(* Logix 5000 project; controller RN21_Architecture 1769-L16ER-BB1B rev 35.11; software revision 35.00; part 4 of 9 *)
(* tags used below, declared in another part *)
   AUDSrc : UDT_Audit;
   RN21_AUD_BAT_NTrig : DINT[4];
   RN21_AUD_BAT_PTrig : DINT[4];
   RN21_AUD_NEG_ONS : BOOL[128];
   RN21_AUD_POS_ONS : BOOL[128];
   RN21_Map_BAT : BOOL[32];
   RN21_MapBAT_OB : BOOL[128];
(* MainProgram, continued *)

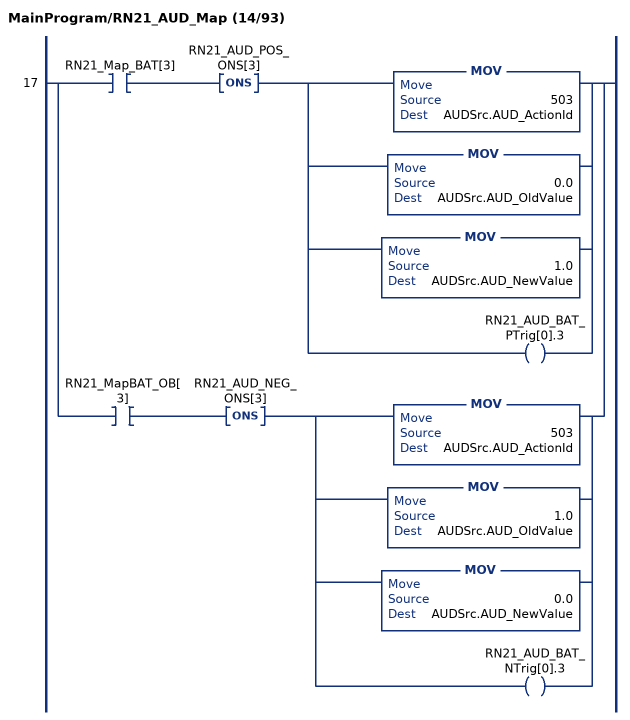
   [picture p96: MainProgram/RN21_AUD_Map rungs 17-17]
   17: [XIC(RN21_Map_BAT[3]) ONS(RN21_AUD_POS_ONS[3]) [MOV(503,AUDSrc.AUD_ActionId) ,MOV(0.0,AUDSrc.AUD_OldValue) ,MOV(1.0,AUDSrc.AUD_NewValue) ,OTE(RN21_AUD_BAT_PTrig[0].3) ] ,XIC(RN21_MapBAT_OB[3]) ONS(RN21_AUD_NEG_ONS[3]) [MOV(503,AUDSrc.AUD_ActionId) ,MOV(1.0,AUDSrc.AUD_OldValue) ,MOV(0.0,AUDSrc.AUD_NewValue) ,OTE(RN21_AUD_BAT_NTrig[0].3) ] ];
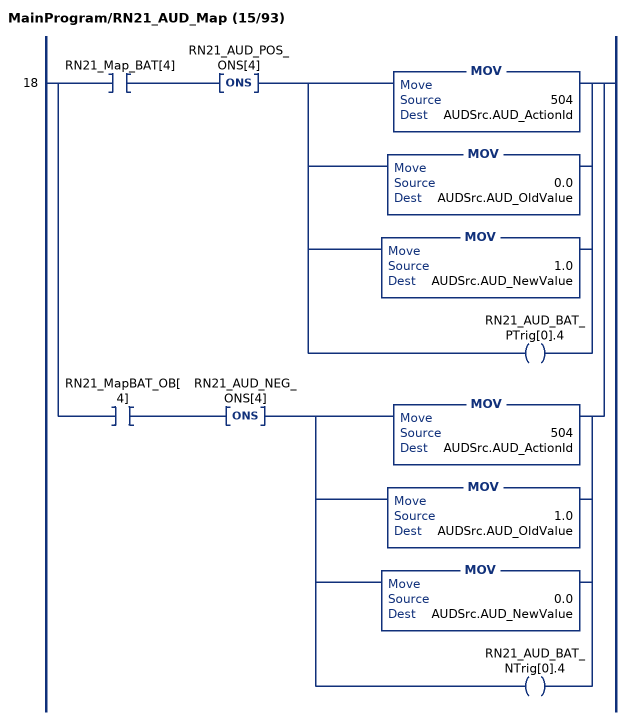
   18: [XIC(RN21_Map_BAT[4]) ONS(RN21_AUD_POS_ONS[4]) [MOV(504,AUDSrc.AUD_ActionId) ,MOV(0.0,AUDSrc.AUD_OldValue) ,MOV(1.0,AUDSrc.AUD_NewValue) ,OTE(RN21_AUD_BAT_PTrig[0].4) ] ,XIC(RN21_MapBAT_OB[4]) ONS(RN21_AUD_NEG_ONS[4]) [MOV(504,AUDSrc.AUD_ActionId) ,MOV(1.0,AUDSrc.AUD_OldValue) ,MOV(0.0,AUDSrc.AUD_NewValue) ,OTE(RN21_AUD_BAT_NTrig[0].4) ] ];
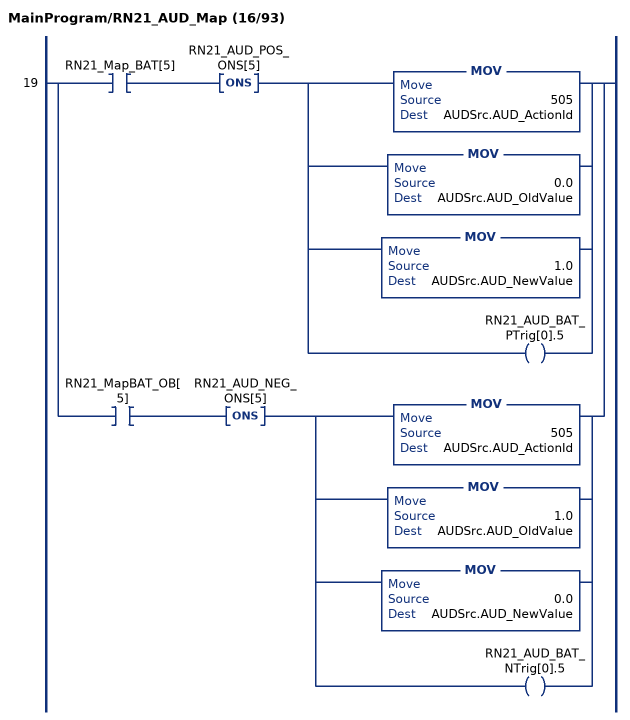
   19: [XIC(RN21_Map_BAT[5]) ONS(RN21_AUD_POS_ONS[5]) [MOV(505,AUDSrc.AUD_ActionId) ,MOV(0.0,AUDSrc.AUD_OldValue) ,MOV(1.0,AUDSrc.AUD_NewValue) ,OTE(RN21_AUD_BAT_PTrig[0].5) ] ,XIC(RN21_MapBAT_OB[5]) ONS(RN21_AUD_NEG_ONS[5]) [MOV(505,AUDSrc.AUD_ActionId) ,MOV(1.0,AUDSrc.AUD_OldValue) ,MOV(0.0,AUDSrc.AUD_NewValue) ,OTE(RN21_AUD_BAT_NTrig[0].5) ] ];
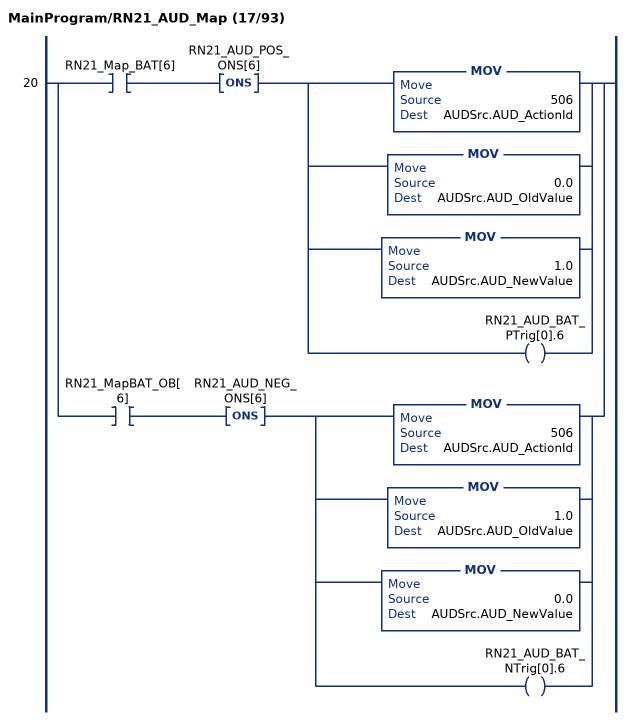
   20: [XIC(RN21_Map_BAT[6]) ONS(RN21_AUD_POS_ONS[6]) [MOV(506,AUDSrc.AUD_ActionId) ,MOV(0.0,AUDSrc.AUD_OldValue) ,MOV(1.0,AUDSrc.AUD_NewValue) ,OTE(RN21_AUD_BAT_PTrig[0].6) ] ,XIC(RN21_MapBAT_OB[6]) ONS(RN21_AUD_NEG_ONS[6]) [MOV(506,AUDSrc.AUD_ActionId) ,MOV(1.0,AUDSrc.AUD_OldValue) ,MOV(0.0,AUDSrc.AUD_NewValue) ,OTE(RN21_AUD_BAT_NTrig[0].6) ] ];
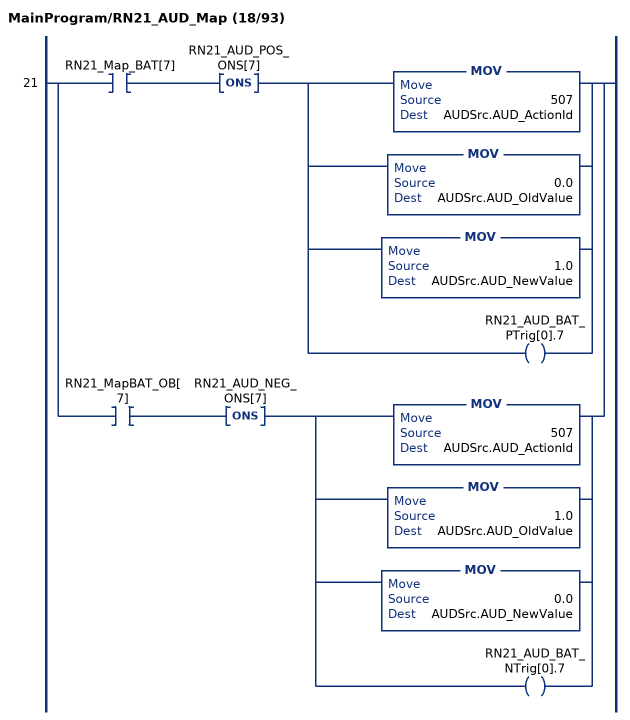
   21: [XIC(RN21_Map_BAT[7]) ONS(RN21_AUD_POS_ONS[7]) [MOV(507,AUDSrc.AUD_ActionId) ,MOV(0.0,AUDSrc.AUD_OldValue) ,MOV(1.0,AUDSrc.AUD_NewValue) ,OTE(RN21_AUD_BAT_PTrig[0].7) ] ,XIC(RN21_MapBAT_OB[7]) ONS(RN21_AUD_NEG_ONS[7]) [MOV(507,AUDSrc.AUD_ActionId) ,MOV(1.0,AUDSrc.AUD_OldValue) ,MOV(0.0,AUDSrc.AUD_NewValue) ,OTE(RN21_AUD_BAT_NTrig[0].7) ] ];
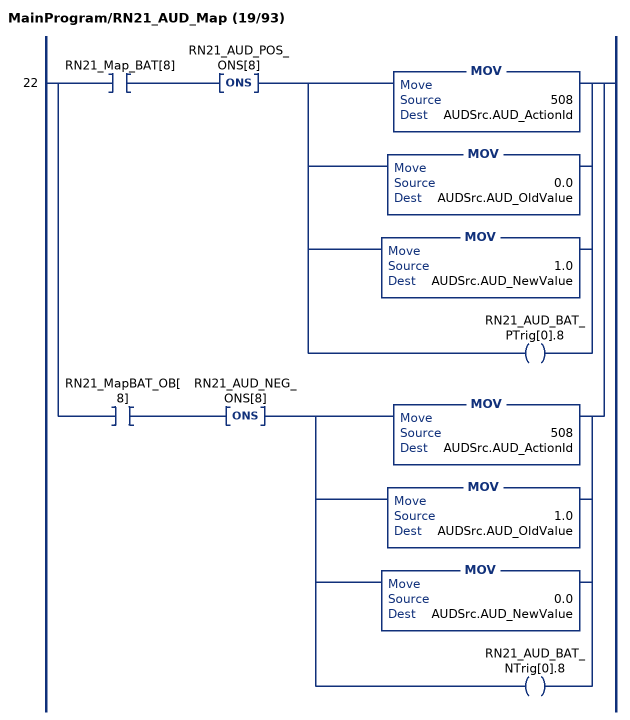
   22: [XIC(RN21_Map_BAT[8]) ONS(RN21_AUD_POS_ONS[8]) [MOV(508,AUDSrc.AUD_ActionId) ,MOV(0.0,AUDSrc.AUD_OldValue) ,MOV(1.0,AUDSrc.AUD_NewValue) ,OTE(RN21_AUD_BAT_PTrig[0].8) ] ,XIC(RN21_MapBAT_OB[8]) ONS(RN21_AUD_NEG_ONS[8]) [MOV(508,AUDSrc.AUD_ActionId) ,MOV(1.0,AUDSrc.AUD_OldValue) ,MOV(0.0,AUDSrc.AUD_NewValue) ,OTE(RN21_AUD_BAT_NTrig[0].8) ] ];
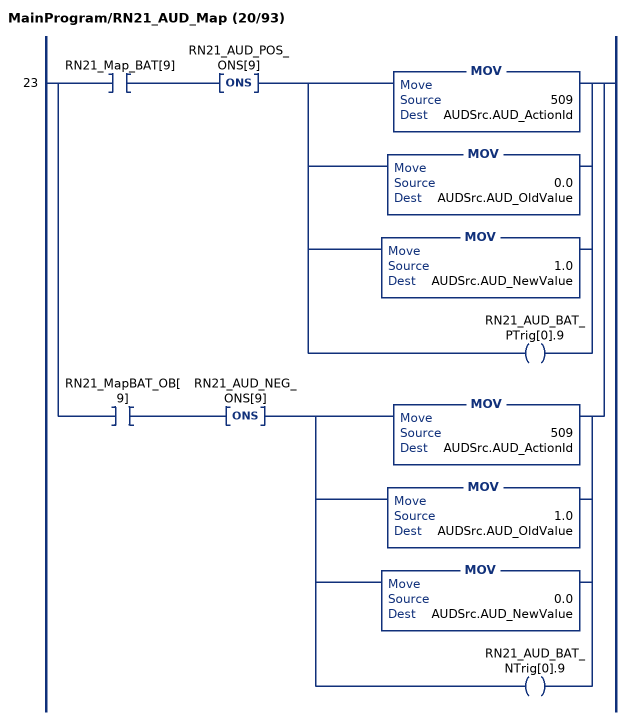
   23: [XIC(RN21_Map_BAT[9]) ONS(RN21_AUD_POS_ONS[9]) [MOV(509,AUDSrc.AUD_ActionId) ,MOV(0.0,AUDSrc.AUD_OldValue) ,MOV(1.0,AUDSrc.AUD_NewValue) ,OTE(RN21_AUD_BAT_PTrig[0].9) ] ,XIC(RN21_MapBAT_OB[9]) ONS(RN21_AUD_NEG_ONS[9]) [MOV(509,AUDSrc.AUD_ActionId) ,MOV(1.0,AUDSrc.AUD_OldValue) ,MOV(0.0,AUDSrc.AUD_NewValue) ,OTE(RN21_AUD_BAT_NTrig[0].9) ] ];
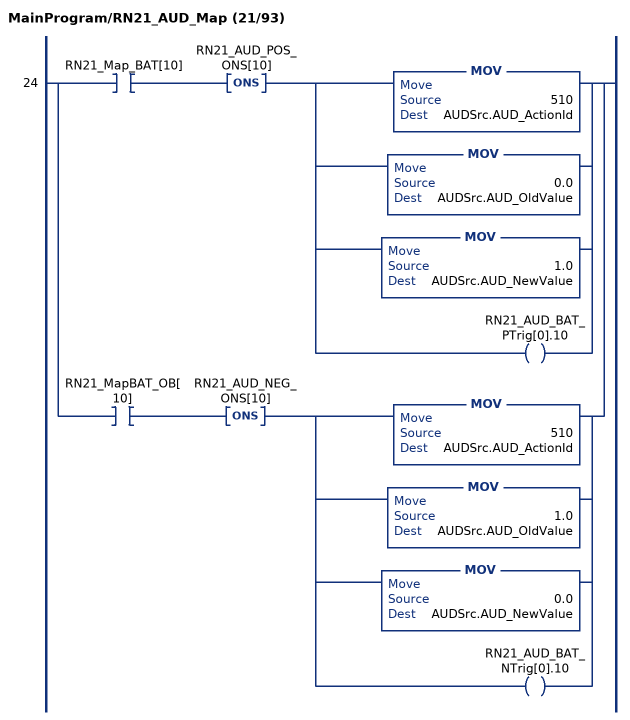
   24: [XIC(RN21_Map_BAT[10]) ONS(RN21_AUD_POS_ONS[10]) [MOV(510,AUDSrc.AUD_ActionId) ,MOV(0.0,AUDSrc.AUD_OldValue) ,MOV(1.0,AUDSrc.AUD_NewValue) ,OTE(RN21_AUD_BAT_PTrig[0].10) ] ,XIC(RN21_MapBAT_OB[10]) ONS(RN21_AUD_NEG_ONS[10]) [MOV(510,AUDSrc.AUD_ActionId) ,MOV(1.0,AUDSrc.AUD_OldValue) ,MOV(0.0,AUDSrc.AUD_NewValue) ,OTE(RN21_AUD_BAT_NTrig[0].10) ] ];
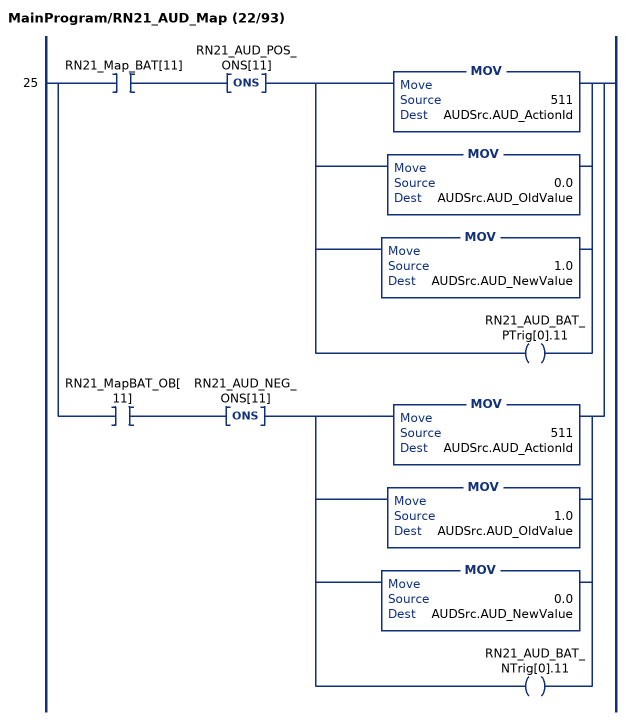
   25: [XIC(RN21_Map_BAT[11]) ONS(RN21_AUD_POS_ONS[11]) [MOV(511,AUDSrc.AUD_ActionId) ,MOV(0.0,AUDSrc.AUD_OldValue) ,MOV(1.0,AUDSrc.AUD_NewValue) ,OTE(RN21_AUD_BAT_PTrig[0].11) ] ,XIC(RN21_MapBAT_OB[11]) ONS(RN21_AUD_NEG_ONS[11]) [MOV(511,AUDSrc.AUD_ActionId) ,MOV(1.0,AUDSrc.AUD_OldValue) ,MOV(0.0,AUDSrc.AUD_NewValue) ,OTE(RN21_AUD_BAT_NTrig[0].11) ] ];
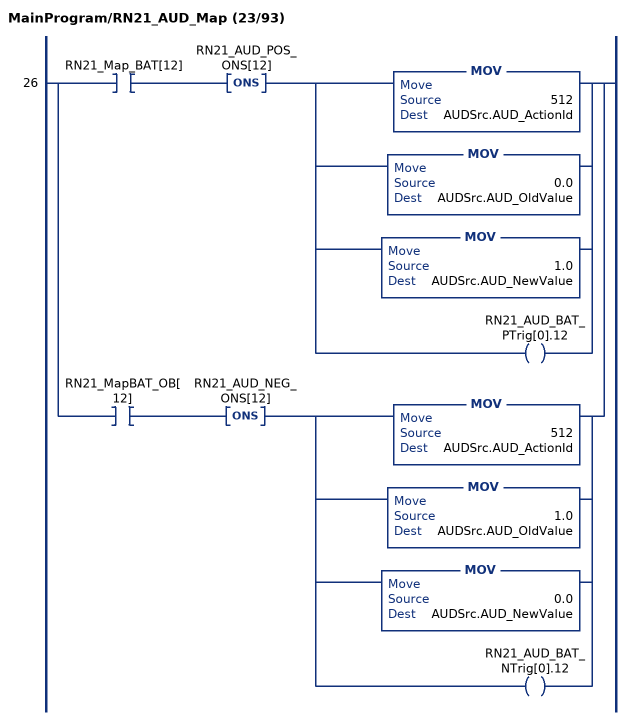
   26: [XIC(RN21_Map_BAT[12]) ONS(RN21_AUD_POS_ONS[12]) [MOV(512,AUDSrc.AUD_ActionId) ,MOV(0.0,AUDSrc.AUD_OldValue) ,MOV(1.0,AUDSrc.AUD_NewValue) ,OTE(RN21_AUD_BAT_PTrig[0].12) ] ,XIC(RN21_MapBAT_OB[12]) ONS(RN21_AUD_NEG_ONS[12]) [MOV(512,AUDSrc.AUD_ActionId) ,MOV(1.0,AUDSrc.AUD_OldValue) ,MOV(0.0,AUDSrc.AUD_NewValue) ,OTE(RN21_AUD_BAT_NTrig[0].12) ] ];
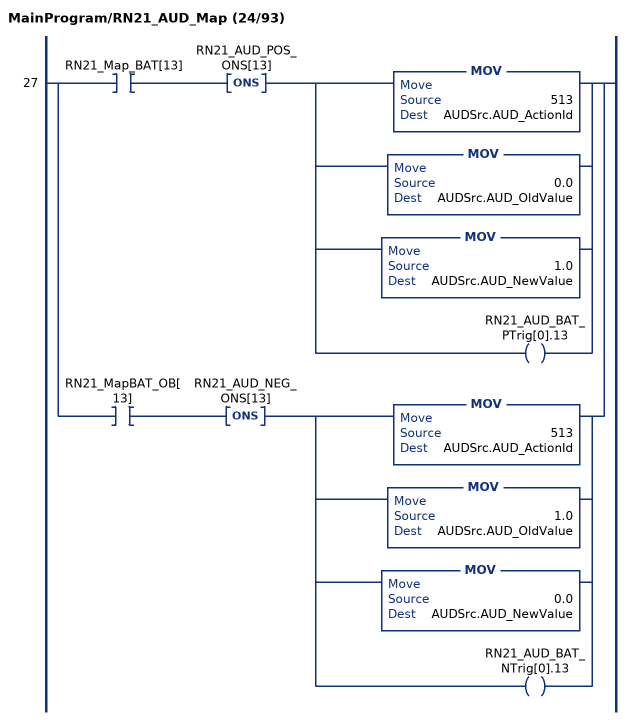
   27: [XIC(RN21_Map_BAT[13]) ONS(RN21_AUD_POS_ONS[13]) [MOV(513,AUDSrc.AUD_ActionId) ,MOV(0.0,AUDSrc.AUD_OldValue) ,MOV(1.0,AUDSrc.AUD_NewValue) ,OTE(RN21_AUD_BAT_PTrig[0].13) ] ,XIC(RN21_MapBAT_OB[13]) ONS(RN21_AUD_NEG_ONS[13]) [MOV(513,AUDSrc.AUD_ActionId) ,MOV(1.0,AUDSrc.AUD_OldValue) ,MOV(0.0,AUDSrc.AUD_NewValue) ,OTE(RN21_AUD_BAT_NTrig[0].13) ] ];
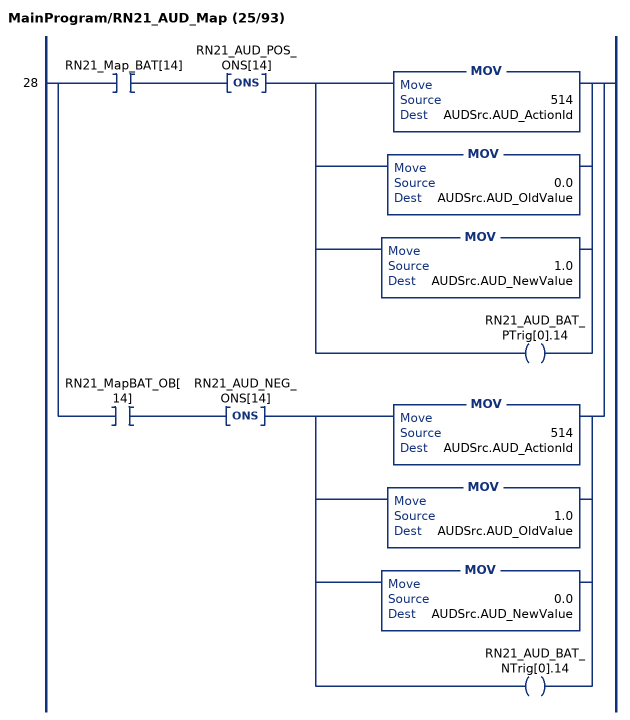
   28: [XIC(RN21_Map_BAT[14]) ONS(RN21_AUD_POS_ONS[14]) [MOV(514,AUDSrc.AUD_ActionId) ,MOV(0.0,AUDSrc.AUD_OldValue) ,MOV(1.0,AUDSrc.AUD_NewValue) ,OTE(RN21_AUD_BAT_PTrig[0].14) ] ,XIC(RN21_MapBAT_OB[14]) ONS(RN21_AUD_NEG_ONS[14]) [MOV(514,AUDSrc.AUD_ActionId) ,MOV(1.0,AUDSrc.AUD_OldValue) ,MOV(0.0,AUDSrc.AUD_NewValue) ,OTE(RN21_AUD_BAT_NTrig[0].14) ] ];
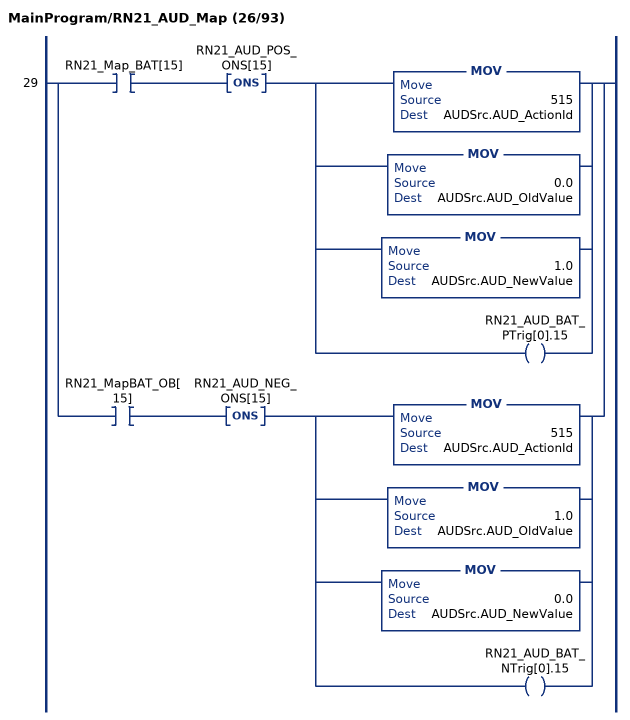
   29: [XIC(RN21_Map_BAT[15]) ONS(RN21_AUD_POS_ONS[15]) [MOV(515,AUDSrc.AUD_ActionId) ,MOV(0.0,AUDSrc.AUD_OldValue) ,MOV(1.0,AUDSrc.AUD_NewValue) ,OTE(RN21_AUD_BAT_PTrig[0].15) ] ,XIC(RN21_MapBAT_OB[15]) ONS(RN21_AUD_NEG_ONS[15]) [MOV(515,AUDSrc.AUD_ActionId) ,MOV(1.0,AUDSrc.AUD_OldValue) ,MOV(0.0,AUDSrc.AUD_NewValue) ,OTE(RN21_AUD_BAT_NTrig[0].15) ] ];
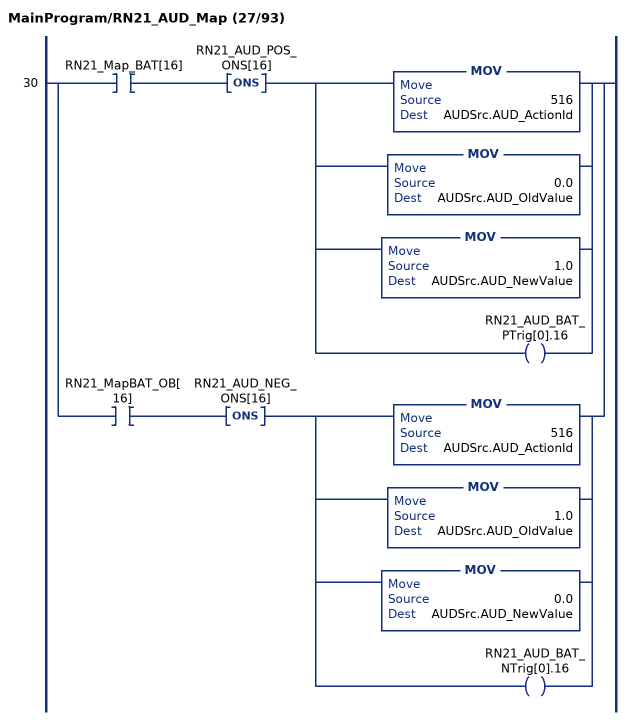
   30: [XIC(RN21_Map_BAT[16]) ONS(RN21_AUD_POS_ONS[16]) [MOV(516,AUDSrc.AUD_ActionId) ,MOV(0.0,AUDSrc.AUD_OldValue) ,MOV(1.0,AUDSrc.AUD_NewValue) ,OTE(RN21_AUD_BAT_PTrig[0].16) ] ,XIC(RN21_MapBAT_OB[16]) ONS(RN21_AUD_NEG_ONS[16]) [MOV(516,AUDSrc.AUD_ActionId) ,MOV(1.0,AUDSrc.AUD_OldValue) ,MOV(0.0,AUDSrc.AUD_NewValue) ,OTE(RN21_AUD_BAT_NTrig[0].16) ] ];
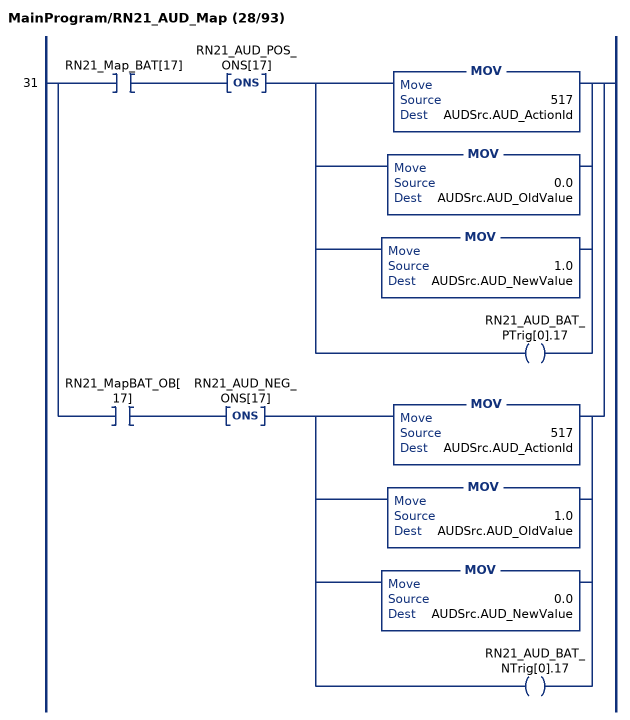
   31: [XIC(RN21_Map_BAT[17]) ONS(RN21_AUD_POS_ONS[17]) [MOV(517,AUDSrc.AUD_ActionId) ,MOV(0.0,AUDSrc.AUD_OldValue) ,MOV(1.0,AUDSrc.AUD_NewValue) ,OTE(RN21_AUD_BAT_PTrig[0].17) ] ,XIC(RN21_MapBAT_OB[17]) ONS(RN21_AUD_NEG_ONS[17]) [MOV(517,AUDSrc.AUD_ActionId) ,MOV(1.0,AUDSrc.AUD_OldValue) ,MOV(0.0,AUDSrc.AUD_NewValue) ,OTE(RN21_AUD_BAT_NTrig[0].17) ] ];
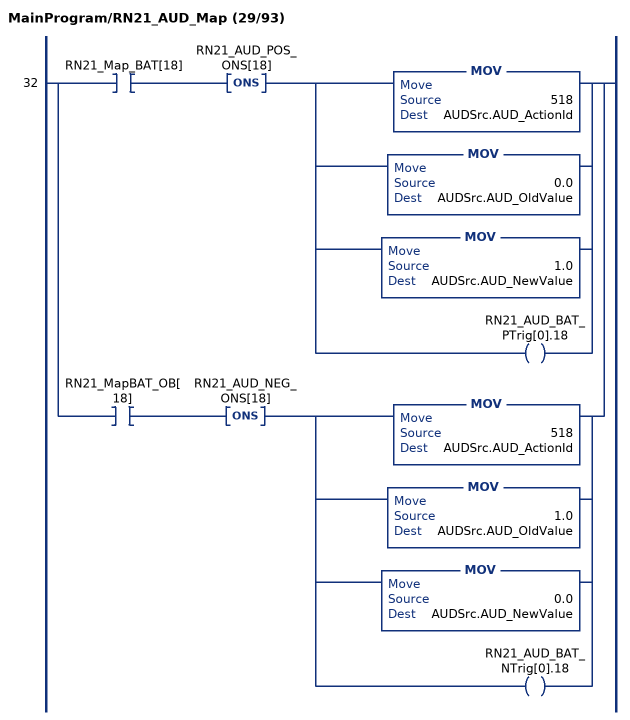
   32: [XIC(RN21_Map_BAT[18]) ONS(RN21_AUD_POS_ONS[18]) [MOV(518,AUDSrc.AUD_ActionId) ,MOV(0.0,AUDSrc.AUD_OldValue) ,MOV(1.0,AUDSrc.AUD_NewValue) ,OTE(RN21_AUD_BAT_PTrig[0].18) ] ,XIC(RN21_MapBAT_OB[18]) ONS(RN21_AUD_NEG_ONS[18]) [MOV(518,AUDSrc.AUD_ActionId) ,MOV(1.0,AUDSrc.AUD_OldValue) ,MOV(0.0,AUDSrc.AUD_NewValue) ,OTE(RN21_AUD_BAT_NTrig[0].18) ] ];
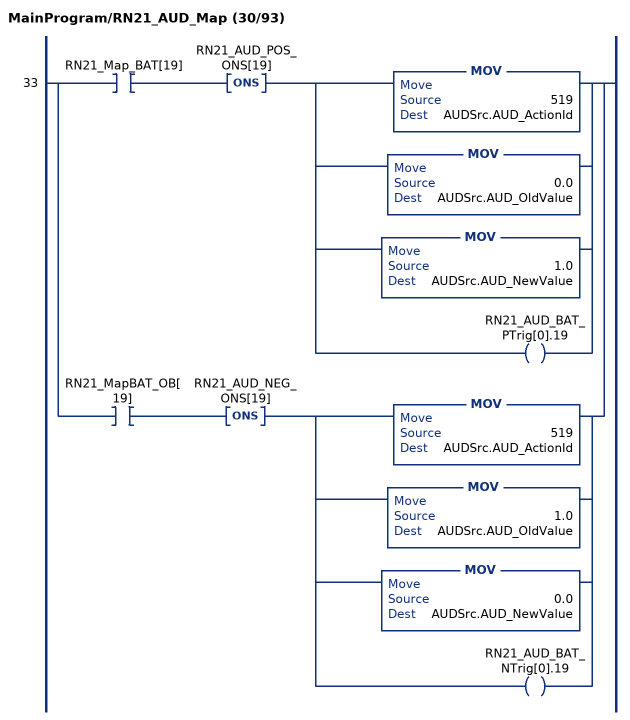
   33: [XIC(RN21_Map_BAT[19]) ONS(RN21_AUD_POS_ONS[19]) [MOV(519,AUDSrc.AUD_ActionId) ,MOV(0.0,AUDSrc.AUD_OldValue) ,MOV(1.0,AUDSrc.AUD_NewValue) ,OTE(RN21_AUD_BAT_PTrig[0].19) ] ,XIC(RN21_MapBAT_OB[19]) ONS(RN21_AUD_NEG_ONS[19]) [MOV(519,AUDSrc.AUD_ActionId) ,MOV(1.0,AUDSrc.AUD_OldValue) ,MOV(0.0,AUDSrc.AUD_NewValue) ,OTE(RN21_AUD_BAT_NTrig[0].19) ] ];
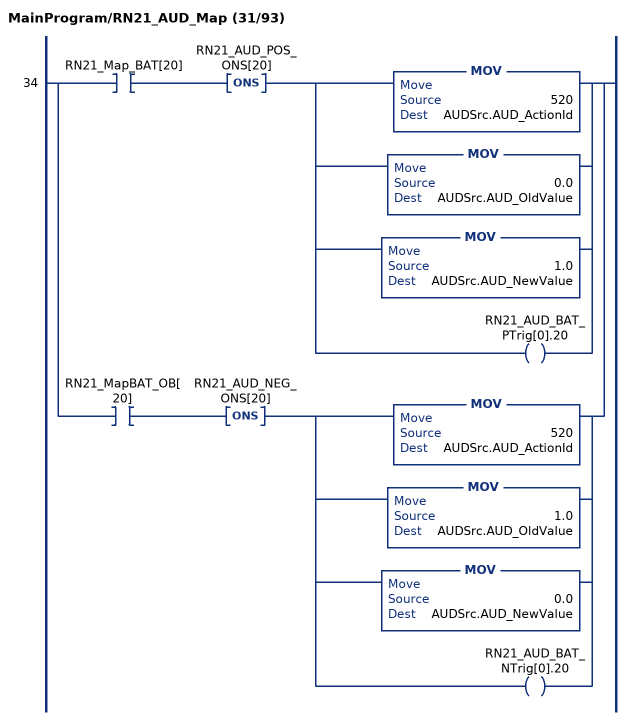
   34: [XIC(RN21_Map_BAT[20]) ONS(RN21_AUD_POS_ONS[20]) [MOV(520,AUDSrc.AUD_ActionId) ,MOV(0.0,AUDSrc.AUD_OldValue) ,MOV(1.0,AUDSrc.AUD_NewValue) ,OTE(RN21_AUD_BAT_PTrig[0].20) ] ,XIC(RN21_MapBAT_OB[20]) ONS(RN21_AUD_NEG_ONS[20]) [MOV(520,AUDSrc.AUD_ActionId) ,MOV(1.0,AUDSrc.AUD_OldValue) ,MOV(0.0,AUDSrc.AUD_NewValue) ,OTE(RN21_AUD_BAT_NTrig[0].20) ] ];
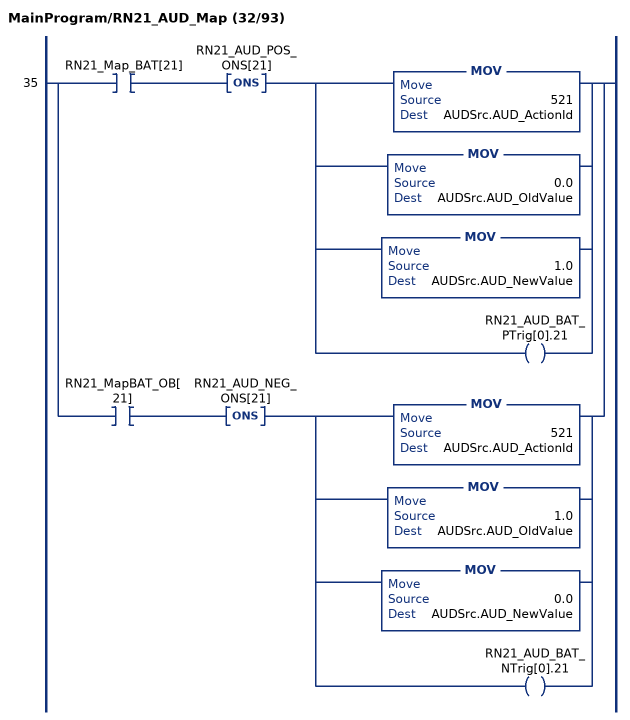
   35: [XIC(RN21_Map_BAT[21]) ONS(RN21_AUD_POS_ONS[21]) [MOV(521,AUDSrc.AUD_ActionId) ,MOV(0.0,AUDSrc.AUD_OldValue) ,MOV(1.0,AUDSrc.AUD_NewValue) ,OTE(RN21_AUD_BAT_PTrig[0].21) ] ,XIC(RN21_MapBAT_OB[21]) ONS(RN21_AUD_NEG_ONS[21]) [MOV(521,AUDSrc.AUD_ActionId) ,MOV(1.0,AUDSrc.AUD_OldValue) ,MOV(0.0,AUDSrc.AUD_NewValue) ,OTE(RN21_AUD_BAT_NTrig[0].21) ] ];
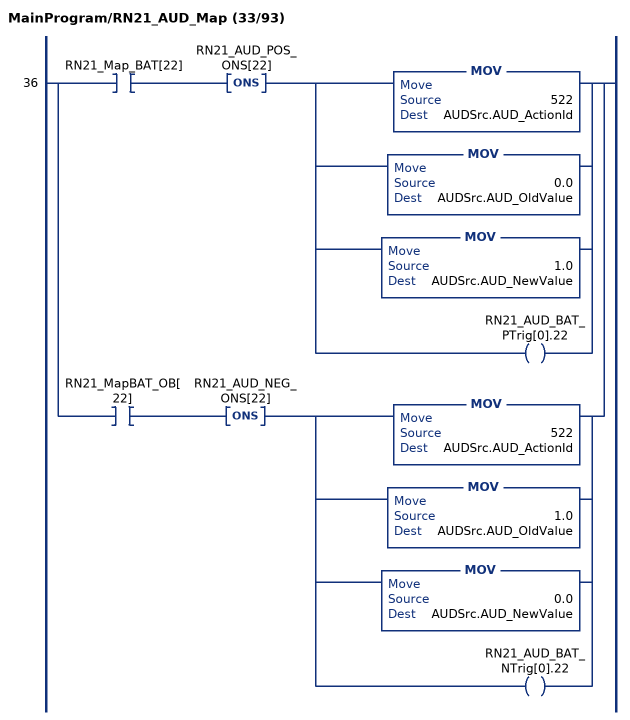
   36: [XIC(RN21_Map_BAT[22]) ONS(RN21_AUD_POS_ONS[22]) [MOV(522,AUDSrc.AUD_ActionId) ,MOV(0.0,AUDSrc.AUD_OldValue) ,MOV(1.0,AUDSrc.AUD_NewValue) ,OTE(RN21_AUD_BAT_PTrig[0].22) ] ,XIC(RN21_MapBAT_OB[22]) ONS(RN21_AUD_NEG_ONS[22]) [MOV(522,AUDSrc.AUD_ActionId) ,MOV(1.0,AUDSrc.AUD_OldValue) ,MOV(0.0,AUDSrc.AUD_NewValue) ,OTE(RN21_AUD_BAT_NTrig[0].22) ] ];
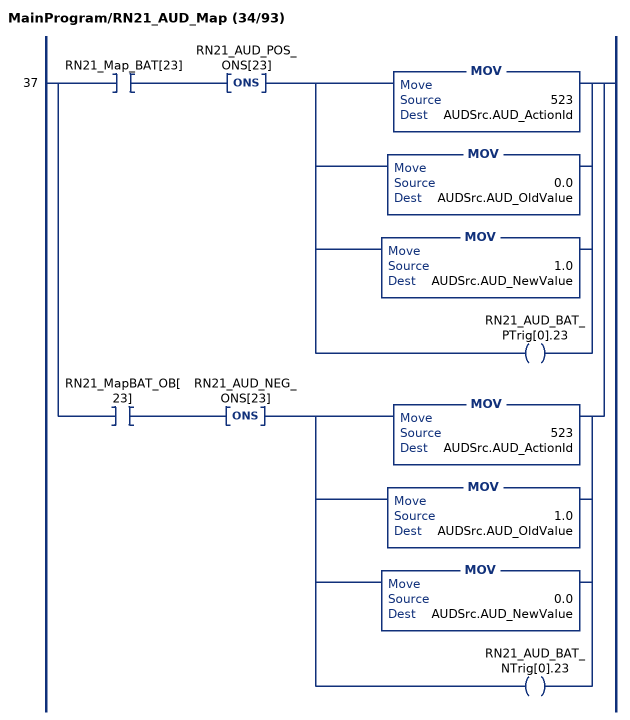
   37: [XIC(RN21_Map_BAT[23]) ONS(RN21_AUD_POS_ONS[23]) [MOV(523,AUDSrc.AUD_ActionId) ,MOV(0.0,AUDSrc.AUD_OldValue) ,MOV(1.0,AUDSrc.AUD_NewValue) ,OTE(RN21_AUD_BAT_PTrig[0].23) ] ,XIC(RN21_MapBAT_OB[23]) ONS(RN21_AUD_NEG_ONS[23]) [MOV(523,AUDSrc.AUD_ActionId) ,MOV(1.0,AUDSrc.AUD_OldValue) ,MOV(0.0,AUDSrc.AUD_NewValue) ,OTE(RN21_AUD_BAT_NTrig[0].23) ] ];
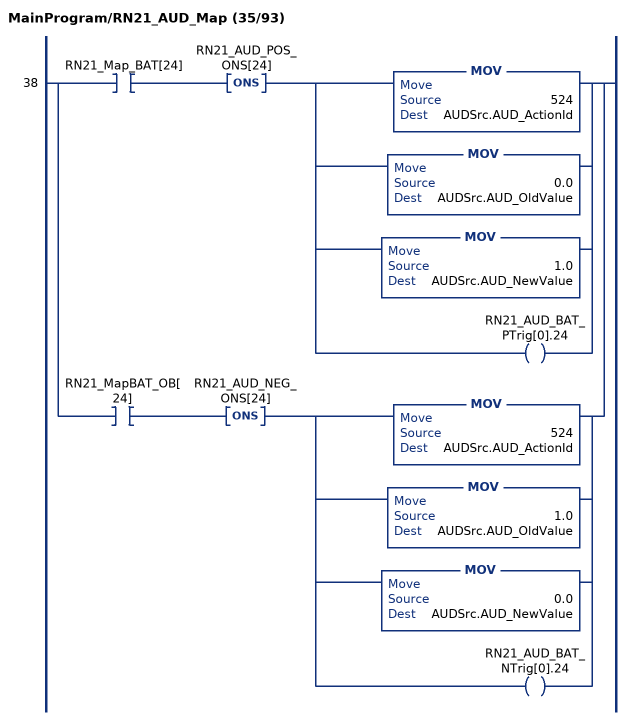
   38: [XIC(RN21_Map_BAT[24]) ONS(RN21_AUD_POS_ONS[24]) [MOV(524,AUDSrc.AUD_ActionId) ,MOV(0.0,AUDSrc.AUD_OldValue) ,MOV(1.0,AUDSrc.AUD_NewValue) ,OTE(RN21_AUD_BAT_PTrig[0].24) ] ,XIC(RN21_MapBAT_OB[24]) ONS(RN21_AUD_NEG_ONS[24]) [MOV(524,AUDSrc.AUD_ActionId) ,MOV(1.0,AUDSrc.AUD_OldValue) ,MOV(0.0,AUDSrc.AUD_NewValue) ,OTE(RN21_AUD_BAT_NTrig[0].24) ] ];
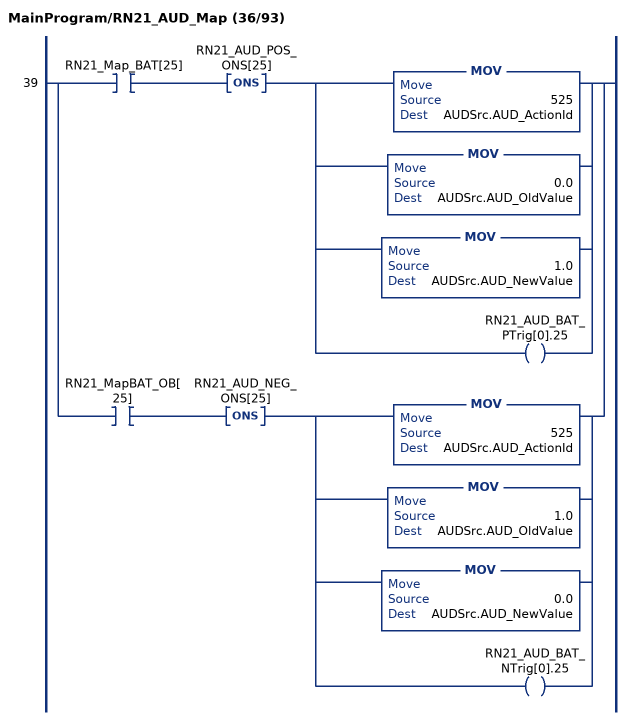
   39: [XIC(RN21_Map_BAT[25]) ONS(RN21_AUD_POS_ONS[25]) [MOV(525,AUDSrc.AUD_ActionId) ,MOV(0.0,AUDSrc.AUD_OldValue) ,MOV(1.0,AUDSrc.AUD_NewValue) ,OTE(RN21_AUD_BAT_PTrig[0].25) ] ,XIC(RN21_MapBAT_OB[25]) ONS(RN21_AUD_NEG_ONS[25]) [MOV(525,AUDSrc.AUD_ActionId) ,MOV(1.0,AUDSrc.AUD_OldValue) ,MOV(0.0,AUDSrc.AUD_NewValue) ,OTE(RN21_AUD_BAT_NTrig[0].25) ] ];
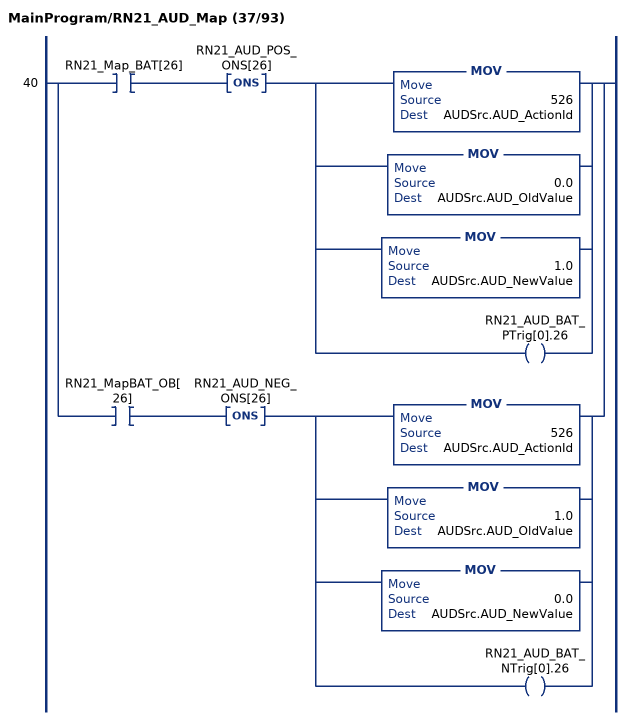
   40: [XIC(RN21_Map_BAT[26]) ONS(RN21_AUD_POS_ONS[26]) [MOV(526,AUDSrc.AUD_ActionId) ,MOV(0.0,AUDSrc.AUD_OldValue) ,MOV(1.0,AUDSrc.AUD_NewValue) ,OTE(RN21_AUD_BAT_PTrig[0].26) ] ,XIC(RN21_MapBAT_OB[26]) ONS(RN21_AUD_NEG_ONS[26]) [MOV(526,AUDSrc.AUD_ActionId) ,MOV(1.0,AUDSrc.AUD_OldValue) ,MOV(0.0,AUDSrc.AUD_NewValue) ,OTE(RN21_AUD_BAT_NTrig[0].26) ] ];
